TYPE E_PickPutMode :
(
	MODE_Pick := 0,
	MODE_Put := 1
)USINT;
END_TYPE

(* stored: Version 1.1.0.1, ProductVersion 3.1.0.25
   DUT E_PickPutMode: Id {cc740aa9-2958-4c7b-9e2e-6e45e2869aed} *)
